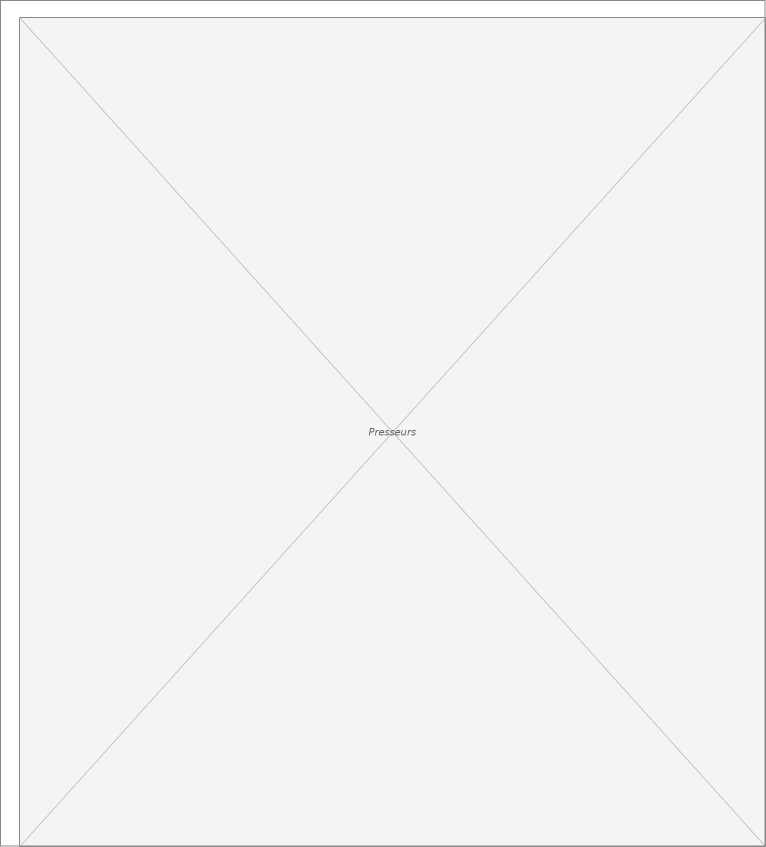
VISUALIZATION Presseurs  // 766x847
    Image (19,17 747x830), image: Presseurs
END_VISUALIZATION

(* stored: Version 1.1.0.1
   Visu Presseurs: Id {d69e81d4-11af-4091-a05b-5a0fbe40cf9b} *)
